    stCoating1 : DUT_PositionState;
    stCoating2 : DUT_PositionState;
END_VAR
VAR_OUTPUT
    {attribute 'pytmc' := '
      pv: GET;
      io: i;
    '}
    enumGet : ENUM_Coating_States;
  END_VAR
VAR
    bCoatingInit : BOOL;
END_VAR

if NOT bCoatingInit THEN
    bCoatingInit := TRUE;

    arrStates[1] := stCoating1;
    arrStates[2] := stCoating2;
END_IF

setState := enumSet;
Exec();
enumGet := getState;
enumSet := setState;

END_FUNCTION_BLOCK

// ---- POUs/Main.TcPOU
PROGRAM Main
VAR
    tpImAPLC : TP := (PT:=T#10S);

    // MR1L3
    // Motors
    {attribute 'TcLinkTo' := '.bLimitForwardEnable:=TIIB[EL7041-1000_M1L3_Yup]^STM Status^Status^Digital input 1;
                              .bLimitBackwardEnable:=TIIB[EL7041-1000_M1L3_Yup]^STM Status^Status^Digital input 2;
                              .nRawEncoderULINT:=TIIB[EL5042_M1L3_Yupdwn]^FB Inputs Channel 1^Position'}
    {attribute 'pytmc' := '
        pv: MR1L3:HOMS:MMS:YUP
    '}
    //PMPS State Stage; bPowerSelf:=False
    M1 : DUT_MotionStage := (sName:='MR1L3-Coatings', fVelocity:=200.0, nEnableMode:=ENUM_StageEnableMode.ALWAYS, bPowerSelf:=FALSE);
    fbMotionStage_m1 : FB_MotionStage;

    {attribute 'TcLinkTo' := '.bLimitForwardEnable:=TIIB[EL7041-1000_M1L3_Ydwn]^STM Status^Status^Digital input 1;
                              .bLimitBackwardEnable:=TIIB[EL7041-1000_M1L3_Ydwn]^STM Status^Status^Digital input 2'}
    {attribute 'pytmc' := '
        pv: MR1L3:HOMS:MMS:YDWN
    '}
    M2 : DUT_MotionStage := (fVelocity:=200.0, nEnableMode:=ENUM_StageEnableMode.ALWAYS, bPowerSelf:=TRUE);
    fbMotionStage_m2 : FB_MotionStage;

    {attribute 'TcLinkTo' := '.bLimitForwardEnable:=TIIB[EL7041-1000_M1L3_Xup]^STM Status^Status^Digital input 1;
                              .bLimitBackwardEnable:=TIIB[EL7041-1000_M1L3_Xup]^STM Status^Status^Digital input 2;
                              .nRawEncoderULINT:=TIIB[EL5042_M1L3_Xupdwn]^FB Inputs Channel 1^Position'}
    {attribute 'pytmc' := '
        pv: MR1L3:HOMS:MMS:XUP
    '}
    M3 : DUT_MotionStage := (fVelocity:=1000.0, nEnableMode:=ENUM_StageEnableMode.ALWAYS, bPowerSelf:=TRUE);
    fbMotionStage_m3 : FB_MotionStage;

    {attribute 'TcLinkTo' := '.bLimitForwardEnable:=TIIB[EL7041-1000_M1L3_Xdwn]^STM Status^Status^Digital input 1;
                              .bLimitBackwardEnable:=TIIB[EL7041-1000_M1L3_Xdwn]^STM Status^Status^Digital input 2'}
    {attribute 'pytmc' := '
        pv: MR1L3:HOMS:MMS:XDWN
    '}
    M4 : DUT_MotionStage := (fVelocity:=1000.0, nEnableMode:=ENUM_StageEnableMode.ALWAYS, bPowerSelf:=TRUE);
    fbMotionStage_m4 : FB_MotionStage;

    {attribute 'TcLinkTo' := '.bLimitForwardEnable:=TIIB[EL7041-1000_M1L3_PitchCoarse]^STM Status^Status^Digital input 1;
                              .bLimitBackwardEnable:=TIIB[EL7041-1000_M1L3_PitchCoarse]^STM Status^Status^Digital input 2;
                              .nRawEncoderULINT:=TIIB[EL5042_M1L3_PitchBender]^FB Inputs Channel 1^Position'}
    {attribute 'pytmc' := '
        pv: MR1L3:HOMS:MMS:PITCH
    '}
    M5 : DUT_MotionStage := (fVelocity:=150.0, nEnableMode:=ENUM_StageEnableMode.ALWAYS, bPowerSelf:=TRUE); // MR1L3 Pitch Stepper
    fbMotionStage_m5 : FB_MotionStage;

    {attribute 'TcLinkTo' := '.bLimitForwardEnable:=TIIB[EL7041-1000_M1L3_Bender]^STM Status^Status^Digital input 1;
                              .bLimitBackwardEnable:=TIIB[EL7041-1000_M1L3_Bender]^STM Status^Status^Digital input 2;
                              .nRawEncoderULINT:=TIIB[EL5042_M1L3_PitchBender]^FB Inputs Channel 2^Position'}
    {attribute 'pytmc' := '
        pv: MR1L3:HOMS:MMS:BENDER
    '}
    M6 : DUT_MotionStage := (fVelocity:=150.0, nEnableMode:=ENUM_StageEnableMode.ALWAYS, bPowerSelf:=TRUE); // MR1L3 Bender
    fbMotionStage_m6 : FB_MotionStage;

    {attribute 'TcLinkTo' := '.fbRunHOMS.bSTOEnable1:=TIIB[EL1004_M1L3_STO]^Channel 1^Input;
                              .fbRunHOMS.bSTOEnable2:=TIIB[EL1004_M1L3_STO]^Channel 2^Input;
                              .fbRunHOMS.stYupEnc.Count:=TIIB[EL5042_M1L3_Yupdwn]^FB Inputs Channel 1^Position;
                              .fbRunHOMS.stYdwnEnc.Count:=TIIB[EL5042_M1L3_Yupdwn]^FB Inputs Channel 2^Position;
                              .fbRunHOMS.stXupEnc.Count:=TIIB[EL5042_M1L3_Xupdwn]^FB Inputs Channel 1^Position;
                              .fbRunHOMS.stXdwnEnc.Count:=TIIB[EL5042_M1L3_Xupdwn]^FB Inputs Channel 2^Position'}
    {attribute 'pytmc' := '
        pv: MR1L3:HOMS
    '}
    MR1L3 : DUT_HOMS;
    {attribute 'pytmc' := '
        pv: MR1L3:HOMS:STATS
    '}
    fbMR1L3GantryStats : FB_HomsStats;

    // Encoder Arrays/RMS Watch:
    {attribute 'pytmc' := '
        pv: MR1L3:HOMS:ENC:Y
    '}
    fbYRMSErrorMR1L3 : FB_RMSWatch;
    fMaxYRMSErrorMR1L3 : LREAL;
    fMinYRMSErrorMR1L3 : LREAL;

    {attribute 'pytmc' := '
        pv: MR1L3:HOMS:ENC:X
    '}
    fbXRMSErrorMR1L3 : FB_RMSWatch;
    fMaxXRMSErrorMR1L3 : LREAL;
    fMinXRMSErrorMR1L3 : LREAL;

    {attribute 'pytmc' := '
        pv: MR1L3:HOMS:ENC:PITCH
    '}
    fbPitchRMSErrorMR1L3 : FB_RMSWatch;
    fMaxPitchRMSErrorMR1L3 : LREAL;
    fMinPitchRMSErrorMR1L3 : LREAL;

    {attribute 'pytmc' := '
        pv: MR1L3:HOMS:ENC:BENDER
    '}
    fbBenderRMSErrorMR1L3 : FB_RMSWatch;
    fMaxBenderRMSErrorMR1L3 : LREAL;
    fMinBenderRMSErrorMR1L3 : LREAL;

    // Pitch Control
    fbMR1L3PitchControl : FB_PitchControl;
    bMR1L3PitchDone : BOOL;
    bMR1L3PitchBusy : BOOL;

    // Bender Control
    fbBenderMR1L3 : FB_Bender;

    // Raw Encoder Counts
    {attribute 'pytmc' := '
        pv: MR1L3:HOMS:ENC:YUP:CNT
        field: EGU cnt
        io: i
    '}
    nEncCntYupMR1L3 : UDINT;
    {attribute 'pytmc' := '
        pv: MR1L3:HOMS:ENC:YDWN:CNT
        field: EGU cnt
        io: i
    '}
    nEncCntYdwnMR1L3 : UDINT;
    {attribute 'pytmc' := '
        pv: MR1L3:HOMS:ENC:XUP:CNT
        field: EGU cnt
        io: i
    '}
    nEncCntXupMR1L3 : UDINT;
    {attribute 'pytmc' := '
        pv: MR1L3:HOMS:ENC:XDWN:CNT
        field: EGU cnt
        io: i
    '}
    nEncCntXdwnMR1L3 : UDINT;
    {attribute 'pytmc' := '
        pv: MR1L3:HOMS:ENC:PITCH:CNT
        field: EGU cnt
        io: i
    '}
    nEncCntPitchMR1L3 : UDINT;

    // Encoder Reference Values
    {attribute 'pytmc' := '
        pv: MR1L3:HOMS:ENC:YUP:REF
        field: EGU cnt
        io: i
    '}
    nEncRefYupMR1L3 : UDINT;
    {attribute 'pytmc' := '
        pv: MR1L3:HOMS:ENC:YDWN:REF
        field: EGU cnt
        io: i
    '}
    nEncRefYdwnMR1L3 : UDINT;
    {attribute 'pytmc' := '
        pv: MR1L3:HOMS:ENC:XUP:REF
        field: EGU cnt
        io: i
    '}
    nEncRefXupMR1L3 : UDINT;
    {attribute 'pytmc' := '
        pv: MR1L3:HOMS:ENC:XDWN:REF
        field: EGU cnt
        io: i
    '}
    nEncRefXdwnMR1L3 : UDINT;
    {attribute 'pytmc' := '
        pv: MR1L3:HOMS:ENC:PITCH:REF
        field: EGU cnt
        io: i
    '}
    nEncRefPitchMR1L3 : UDINT;
    mcReadParameterPitchMR1L3 : MC_ReadParameter;
    fEncRefPitchMR1L3_urad : LREAL; // Current Pitch encoder offset in urad
    // MR1L4
    // Motors
    {attribute 'TcLinkTo' := '.bLimitForwardEnable:=TIIB[EL7041-1000_M1L4_Yup]^STM Status^Status^Digital input 1;
                              .bLimitBackwardEnable:=TIIB[EL7041-1000_M1L4_Yup]^STM Status^Status^Digital input 2;
                              .nRawEncoderULINT:=TIIB[EL5042_M1L4_Yupdwn]^FB Inputs Channel 1^Position'}
    {attribute 'pytmc' := '
        pv: MR1L4:HOMS:MMS:YUP
    '}
    M7 : DUT_MotionStage := (fVelocity:=200.0, nEnableMode:=ENUM_StageEnableMode.ALWAYS, bPowerSelf:=TRUE);
    fbMotionStage_m7 : FB_MotionStage;
    {attribute 'TcLinkTo' := '.bLimitForwardEnable:=TIIB[EL7041-1000_M1L4_Ydwn]^STM Status^Status^Digital input 1;
                              .bLimitBackwardEnable:=TIIB[EL7041-1000_M1L4_Ydwn]^STM Status^Status^Digital input 2'}
    {attribute 'pytmc' := '
        pv: MR1L4:HOMS:MMS:YDWN
    '}
    M8 : DUT_MotionStage := (fVelocity:=200.0, nEnableMode:=ENUM_StageEnableMode.ALWAYS, bPowerSelf:=TRUE);
    fbMotionStage_m8 : FB_MotionStage;
    {attribute 'TcLinkTo' := '.bLimitForwardEnable:=TIIB[EL7041-1000_M1L4_Xup]^STM Status^Status^Digital input 1;
                              .bLimitBackwardEnable:=TIIB[EL7041-1000_M1L4_Xup]^STM Status^Status^Digital input 2;
                              .nRawEncoderULINT:=TIIB[EL5042_M1L4_Xupdwn]^FB Inputs Channel 1^Position'}
    {attribute 'pytmc' := '
        pv: MR1L4:HOMS:MMS:XUP
    '}
    M9 : DUT_MotionStage := (fVelocity:=1000.0, nEnableMode:=ENUM_StageEnableMode.ALWAYS, bPowerSelf:=TRUE);
    fbMotionStage_m9 : FB_MotionStage;
    {attribute 'TcLinkTo' := '.bLimitForwardEnable:=TIIB[EL7041-1000_M1L4_Xdwn]^STM Status^Status^Digital input 1;
                              .bLimitBackwardEnable:=TIIB[EL7041-1000_M1L4_Xdwn]^STM Status^Status^Digital input 2'}
    {attribute 'pytmc' := '
        pv: MR1L4:HOMS:MMS:XDWN
    '}
    M10 : DUT_MotionStage := (fVelocity:=1000.0, nEnableMode:=ENUM_StageEnableMode.ALWAYS, bPowerSelf:=TRUE);
    fbMotionStage_m10 : FB_MotionStage;
    {attribute 'TcLinkTo' := '.bLimitForwardEnable:=TIIB[EL7041-1000_M1L4_PitchCoarse]^STM Status^Status^Digital input 1;
                              .bLimitBackwardEnable:=TIIB[EL7041-1000_M1L4_PitchCoarse]^STM Status^Status^Digital input 2;
                              .nRawEncoderULINT:=TIIB[EL5042_M1L4_PitchBender]^FB Inputs Channel 1^Position'}
    {attribute 'pytmc' := '
        pv: MR1L4:HOMS:MMS:PITCH
    '}
    M11 : DUT_MotionStage := (fVelocity:=150.0, nEnableMode:=ENUM_StageEnableMode.ALWAYS, bPowerSelf:=TRUE); // MR1L4 Pitch Stepper
    fbMotionStage_m11 : FB_MotionStage;
    {attribute 'TcLinkTo' := '.bLimitForwardEnable:=TIIB[EL7041-1000_M1L4_Bender]^STM Status^Status^Digital input 1;
                              .bLimitBackwardEnable:=TIIB[EL7041-1000_M1L4_Bender]^STM Status^Status^Digital input 2;
                              .nRawEncoderULINT:=TIIB[EL5042_M1L4_PitchBender]^FB Inputs Channel 2^Position'}
    {attribute 'pytmc' := '
        pv: MR1L4:HOMS:MMS:BENDER
    '}
    M12 : DUT_MotionStage := (fVelocity:=150.0, nEnableMode:=ENUM_StageEnableMode.ALWAYS, bPowerSelf:=TRUE); // MR1L4 Bender
    fbMotionStage_m12 : FB_MotionStage;
    {attribute 'TcLinkTo' := '.fbRunHOMS.bSTOEnable1:=TIIB[EL1004_M1L4_STO]^Channel 1^Input;
                              .fbRunHOMS.bSTOEnable2:=TIIB[EL1004_M1L4_STO]^Channel 2^Input;
                              .fbRunHOMS.stYupEnc.Count:=TIIB[EL5042_M1L4_Yupdwn]^FB Inputs Channel 1^Position;
                              .fbRunHOMS.stYdwnEnc.Count:=TIIB[EL5042_M1L4_Yupdwn]^FB Inputs Channel 2^Position;
                              .fbRunHOMS.stXupEnc.Count:=TIIB[EL5042_M1L4_Xupdwn]^FB Inputs Channel 1^Position;
                              .fbRunHOMS.stXdwnEnc.Count:=TIIB[EL5042_M1L4_Xupdwn]^FB Inputs Channel 2^Position'}
    {attribute 'pytmc' := '
        pv: MR1L4:HOMS
    '}
    MR1L4 : DUT_HOMS;
    {attribute 'pytmc' := '
        pv: MR1L4:HOMS:STATS
    '}
    fbMR1L4GantryStats : FB_HomsStats;
    // Encoder Arrays/RMS Watch:
    {attribute 'pytmc' := '
        pv: MR1L4:HOMS:ENC:Y
    '}
    fbYRMSErrorMR1L4 : FB_RMSWatch;
    fMaxYRMSErrorMR1L4 : LREAL;
    fMinYRMSErrorMR1L4 : LREAL;

    {attribute 'pytmc' := '
        pv: MR1L4:HOMS:ENC:X
    '}
    fbXRMSErrorMR1L4 : FB_RMSWatch;
    fMaxXRMSErrorMR1L4 : LREAL;
    fMinXRMSErrorMR1L4 : LREAL;

    {attribute 'pytmc' := '
        pv: MR1L4:HOMS:ENC:PITCH
    '}
    fbPitchRMSErrorMR1L4 : FB_RMSWatch;
    fMaxPitchRMSErrorMR1L4 : LREAL;
    fMinPitchRMSErrorMR1L4 : LREAL;

    {attribute 'pytmc' := '
        pv: MR1L4:HOMS:ENC:BENDER
    '}
    fbBenderRMSErrorMR1L4 : FB_RMSWatch;
    fMaxBenderRMSErrorMR1L4 : LREAL;
    fMinBenderRMSErrorMR1L4 : LREAL;

    // Pitch Control
    fbMR1L4PitchControl : FB_PitchControl;
    bMR1L4PitchDone : BOOL;
    bMR1L4PitchBusy : BOOL;

    // Bender Control
    fbBenderMR1L4 : FB_Bender;

    // Raw Encoder Counts
    {attribute 'pytmc' := '
        pv: MR1L4:HOMS:ENC:YUP:CNT
        field: EGU cnt
        io: i
    '}
    nEncCntYupMR1L4 : UDINT;
    {attribute 'pytmc' := '
        pv: MR1L4:HOMS:ENC:YDWN:CNT
        field: EGU cnt
        io: i
    '}
    nEncCntYdwnMR1L4 : UDINT;
    {attribute 'pytmc' := '
        pv: MR1L4:HOMS:ENC:XUP:CNT
        field: EGU cnt
        io: i
    '}
    nEncCntXupMR1L4 : UDINT;
    {attribute 'pytmc' := '
        pv: MR1L4:HOMS:ENC:XDWN:CNT
        field: EGU cnt
        io: i
    '}
    nEncCntXdwnMR1L4 : UDINT;
    {attribute 'pytmc' := '
        pv: MR1L4:HOMS:ENC:PITCH:CNT
        field: EGU cnt
        io: i
    '}
    nEncCntPitchMR1L4 : UDINT;

    // Encoder Reference Values
    {attribute 'pytmc' := '
        pv: MR1L4:HOMS:ENC:YUP:REF
        field: EGU cnt
        io: i
    '}
    nEncRefYupMR1L4 : UDINT;
    {attribute 'pytmc' := '
        pv: MR1L4:HOMS:ENC:YDWN:REF
        field: EGU cnt
        io: i
    '}
    nEncRefYdwnMR1L4 : UDINT;
    {attribute 'pytmc' := '
        pv: MR1L4:HOMS:ENC:XUP:REF
        field: EGU cnt
        io: i
    '}
    nEncRefXupMR1L4 : UDINT;
    {attribute 'pytmc' := '
        pv: MR1L4:HOMS:ENC:XDWN:REF
        field: EGU cnt
        io: i
    '}
    nEncRefXdwnMR1L4 : UDINT;
    {attribute 'pytmc' := '
        pv: MR1L4:HOMS:ENC:PITCH:REF
        field: EGU cnt
        io: i
    '}
    nEncRefPitchMR1L4 : UDINT;
    mcReadParameterPitchMR1L4 : MC_ReadParameter;
    fEncRefPitchMR1L4_urad : LREAL; // Current Pitch encoder offset in urad

// MR2L3 BECKHOFF
// Motors
    {attribute 'TcLinkTo' := '.bLimitForwardEnable:=TIIB[EL7041-1000_M2L3_Yup]^STM Status^Status^Digital input 1;
                              .bLimitBackwardEnable:=TIIB[EL7041-1000_M2L3_Yup]^STM Status^Status^Digital input 2';
                              .nRawEncoderULINT:=TIIB[EL5042_M2L3_Yupdwn]^FB Inputs Channel 1^Position'}
    {attribute 'pytmc' := '
        pv: MR2L3:HOMS:MMS:YUP
    '}
    M13 : DUT_MotionStage := (fVelocity:=200.0, nEnableMode:=ENUM_StageEnableMode.ALWAYS, bPowerSelf:=TRUE); // MR2L3 Yup
    fbMotionStage_m13 : FB_MotionStage;


    {attribute 'TcLinkTo' := '.bLimitForwardEnable:=TIIB[EL7041-1000_M2L3_Ydwn]^STM Status^Status^Digital input 1;
                              .bLimitBackwardEnable:=TIIB[EL7041-1000_M2L3_Ydwn]^STM Status^Status^Digital input 2'}
    {attribute 'pytmc' := '
        pv: MR2L3:HOMS:MMS:YDWN
    '}
    M14 : DUT_MotionStage := (fVelocity:=200.0, nEnableMode:=ENUM_StageEnableMode.ALWAYS, bPowerSelf:=TRUE); // MR2L3 Ydwn
    fbMotionStage_m14 : FB_MotionStage;

    {attribute 'TcLinkTo' := '.bLimitForwardEnable:=TIIB[EL7041-1000_M2L3_Xup]^STM Status^Status^Digital input 1;
                              .bLimitBackwardEnable:=TIIB[EL7041-1000_M2L3_Xup]^STM Status^Status^Digital input 2;
                              .nRawEncoderULINT:=TIIB[EL5042_M2L3_Xupdwn]^FB Inputs Channel 1^Position'}
    {attribute 'pytmc' := '
        pv: MR2L3:HOMS:MMS:XUP
    '}
    M15 : DUT_MotionStage := (fVelocity:=1000.0, nEnableMode:=ENUM_StageEnableMode.ALWAYS, bPowerSelf:=TRUE); // MR2L3 Xup
    fbMotionStage_m15 : FB_MotionStage;

    {attribute 'TcLinkTo' := '.bLimitForwardEnable:=TIIB[EL7041-1000_M2L3_Xdwn]^STM Status^Status^Digital input 1;
                              .bLimitBackwardEnable:=TIIB[EL7041-1000_M2L3_Xdwn]^STM Status^Status^Digital input 2'}
    {attribute 'pytmc' := '
        pv: MR2L3:HOMS:MMS:XDWN
    '}
    M16 : DUT_MotionStage := (fVelocity:=1000.0, nEnableMode:=ENUM_StageEnableMode.ALWAYS, bPowerSelf:=TRUE); // MR2L3 Xdwn
    fbMotionStage_m16 : FB_MotionStage;

    {attribute 'TcLinkTo' := '.bLimitForwardEnable:=TIIB[EL7041-1000_M2L3_PitchCoarse]^STM Status^Status^Digital input 1;
                              .bLimitBackwardEnable:=TIIB[EL7041-1000_M2L3_PitchCoarse]^STM Status^Status^Digital input 2;
                              .nRawEncoderULINT:=TIIB[EL5042_M2L3_PitchBender]^FB Inputs Channel 1^Position'}
    {attribute 'pytmc' := '
        pv: MR2L3:HOMS:MMS:PITCH
    '}
    M17 : DUT_MotionStage := (fVelocity:=150.0, nEnableMode:=ENUM_StageEnableMode.ALWAYS, bPowerSelf:=TRUE); // MR2L3 Pitch Stepper
    fbMotionStage_m17 : FB_MotionStage;
    {attribute 'TcLinkTo' := '.bLimitForwardEnable:=TIIB[EL7041-1000_M2L3_Bender]^STM Status^Status^Digital input 1;
                              .bLimitBackwardEnable:=TIIB[EL7041-1000_M2L3_Bender]^STM Status^Status^Digital input 2;
                              .nRawEncoderULINT:=TIIB[EL5042_M2L3_PitchBender]^FB Inputs Channel 2^Position'}
    {attribute 'pytmc' := '
        pv: MR2L3:HOMS:MMS:BENDER
    '}
    M18 : DUT_MotionStage := (fVelocity:=150.0, nEnableMode:=ENUM_StageEnableMode.ALWAYS, bPowerSelf:=TRUE); // MR2L3 Bender
    fbMotionStage_m18 : FB_MotionStage;

    {attribute 'TcLinkTo' := '.fbRunHOMS.bSTOEnable1:=TIIB[EL1004_M2L3_STO]^Channel 1^Input;
                              .fbRunHOMS.bSTOEnable2:=TIIB[EL1004_M2L3_STO]^Channel 2^Input;
                              .fbRunHOMS.stYupEnc.Count:=TIIB[EL5042_M2L3_Yupdwn]^FB Inputs Channel 1^Position;
                              .fbRunHOMS.stYdwnEnc.Count:=TIIB[EL5042_M2L3_Yupdwn]^FB Inputs Channel 2^Position;
                              .fbRunHOMS.stXupEnc.Count:=TIIB[EL5042_M2L3_Xupdwn]^FB Inputs Channel 1^Position;
                              .fbRunHOMS.stXdwnEnc.Count:=TIIB[EL5042_M2L3_Xupdwn]^FB Inputs Channel 2^Position'}
    {attribute 'pytmc' := '
        pv: MR2L3:HOMS
    '}
    MR2L3 : DUT_HOMS;
    {attribute 'pytmc' := '
        pv: MR2L3:HOMS:STATS
    '}
    fbMR2L3GantryStats : FB_HomsStats;

    // Encoder Arrays/RMS Watch:
    {attribute 'pytmc' := '
        pv: MR2L3:HOMS:ENC:Y
    '}
    fbYRMSErrorMR2L3 : FB_RMSWatch;
    fMaxYRMSErrorMR2L3 : LREAL;
    fMinYRMSErrorMR2L3 : LREAL;

    {attribute 'pytmc' := '
        pv: MR2L3:HOMS:ENC:X
    '}
    fbXRMSErrorMR2L3 : FB_RMSWatch;
    fMaxXRMSErrorMR2L3 : LREAL;
    fMinXRMSErrorMR2L3 : LREAL;

    {attribute 'pytmc' := '
        pv: MR2L3:HOMS:ENC:PITCH
    '}
    fbPitchRMSErrorMR2L3 : FB_RMSWatch;
    fMaxPitchRMSErrorMR2L3 : LREAL;
    fMinPitchRMSErrorMR2L3 : LREAL;

    {attribute 'pytmc' := '
        pv: MR2L3:HOMS:ENC:BENDER
    '}
    fbBenderRMSErrorMR2L3 : FB_RMSWatch;
    fMaxBenderRMSErrorMR2L3 : LREAL;
    fMinBenderRMSErrorMR2L3 : LREAL;

    // Pitch Control
    fbMR2L3PitchControl : FB_PitchControl;
    bMR2L3PitchDone : BOOL;
    bMR2L3PitchBusy : BOOL;

    // Bender Control
    fbBenderMR2L3 : FB_Bender;

    // Raw Encoder Counts
    {attribute 'pytmc' := '
        pv: MR2L3:HOMS:ENC:YUP:CNT
        field: EGU cnt
        io: i
    '}
    nEncCntYupMR2L3 : UDINT;
    {attribute 'pytmc' := '
        pv: MR2L3:HOMS:ENC:YDWN:CNT
        field: EGU cnt
        io: i
    '}
    nEncCntYdwnMR2L3 : UDINT;
    {attribute 'pytmc' := '
        pv: MR2L3:HOMS:ENC:XUP:CNT
        field: EGU cnt
        io: i
    '}
    nEncCntXupMR2L3 : UDINT;
    {attribute 'pytmc' := '
        pv: MR2L3:HOMS:ENC:XDWN:CNT
        field: EGU cnt
        io: i
    '}
    nEncCntXdwnMR2L3 : UDINT;
    {attribute 'pytmc' := '
        pv: MR2L3:HOMS:ENC:PITCH:CNT
        field: EGU cnt
        io: i
    '}
    nEncCntPitchMR2L3 : UDINT;

    // Encoder Reference Values
    {attribute 'pytmc' := '
        pv: MR2L3:HOMS:ENC:YUP:REF
        field: EGU cnt
        io: i
    '}
    nEncRefYupMR2L3 : UDINT;
    {attribute 'pytmc' := '
        pv: MR2L3:HOMS:ENC:YDWN:REF
        field: EGU cnt
        io: i
    '}
    nEncRefYdwnMR2L3 : UDINT;
    {attribute 'pytmc' := '
        pv: MR2L3:HOMS:ENC:XUP:REF
        field: EGU cnt
        io: i
    '}
    nEncRefXupMR2L3 : UDINT;
    {attribute 'pytmc' := '
        pv: MR2L3:HOMS:ENC:XDWN:REF
        field: EGU cnt
        io: i
    '}
    nEncRefXdwnMR2L3 : UDINT;
    {attribute 'pytmc' := '
        pv: MR2L3:HOMS:ENC:PITCH:REF
        field: EGU cnt
        io: i
    '}
    nEncRefPitchMR2L3 : UDINT;
    mcReadParameterPitchMR2L3 : MC_ReadParameter;
    fEncRefPitchMR2L3_urad : LREAL; // Current Pitch encoder offset in urad


    // Common
    fEncLeverArm_mm : LREAL := 513.0;

    // Logging
    fbLogHandler : FB_LogHandler;
END_VAR

// MR1L3 BECKHOFF
MR1L3.fbRunHOMS(stYup:=M1,
               stYdwn:=M2,
               stXup:=M3,
               stXdwn:=M4,
               stPitch:=M5,
               nYupEncRef:=GVL_MR1L3_Constants.nYUP_ENC_REF,
               nYdwnEncRef:=GVL_MR1L3_Constants.nYDWN_ENC_REF,
               nXupEncRef:=GVL_MR1L3_Constants.nXUP_ENC_REF,
               nXdwnEncRef:=GVL_MR1L3_Constants.nXDWN_ENC_REF,
               bExecuteCoupleY:=MR1L3.bExecuteCoupleY,
               bExecuteCoupleX:=MR1L3.bExecuteCoupleX,
               bExecuteDecoupleY:=MR1L3.bExecuteDecoupleY,
               bExecuteDecoupleX:=MR1L3.bExecuteDecoupleX,
               bGantryAlreadyCoupledY=>MR1L3.bGantryAlreadyCoupledY,
               bGantryAlreadyCoupledX=>MR1L3.bGantryAlreadyCoupledX,
               nCurrGantryY=>MR1L3.nCurrGantryY,
               nCurrGantryX=>MR1L3.nCurrGantryX);
fbBenderMR1L3(stBender:=M6,
             bSTOEnable1:=MR1L3.fbRunHOMS.bSTOEnable1,
             bSTOEnable2:=MR1L3.fbRunHOMS.bSTOEnable2);
// No slave motion through Epics
M2.bExecute := FALSE; // MR1L3-Ydwn
M4.bExecute := FALSE; // MR1L3-Xdwn

// Convert nCurrGantry to um (smaller number) to read out in epics
MR1L3.fCurrGantryY_um := LINT_TO_REAL(MR1L3.nCurrGantryY) / 1000.0;
MR1L3.fCurrGantryX_um := LINT_TO_REAL(MR1L3.nCurrGantryX) / 1000.0;

// FB_MotionStage's for non-piezo axes
fbMotionStage_m1(stMotionStage:=M1);
fbMotionStage_m2(stMotionStage:=M2);
fbMotionStage_m3(stMotionStage:=M3);
fbMotionStage_m4(stMotionStage:=M4);
fbMotionStage_m5(stMotionStage:=M5);
fbMotionStage_m6(stMotionStage:=M6);

// Calculate Gantry Stats
fbMR1L3GantryStats(homs:=MR1L3, fbUpStreamY:=M1, fbUpStreamX:=M3);
fbMR1L4GantryStats(homs:=MR1L4, fbUpStreamY:=M7, fbUpStreamX:=M9);
fbMR2L3GantryStats(homs:=MR2L3, fbUpStreamY:=M13, fbUpStreamX:=M15);

// Calculate Pitch RMS Error:
fbYRMSErrorMR1L3(stMotionStage:=M1,
                fMaxRMSError=>fMaxYRMSErrorMR1L3,
                fMinRMSError=>fMinYRMSErrorMR1L3);

fbXRMSErrorMR1L3(stMotionStage:=M3,
                fMaxRMSError=>fMaxXRMSErrorMR1L3,
                fMinRMSError=>fMinXRMSErrorMR1L3);

fbPitchRMSErrorMR1L3(stMotionStage:=M5,
                    fMaxRMSError=>fMaxPitchRMSErrorMR1L3,
                    fMinRMSError=>fMinPitchRMSErrorMR1L3);

fbBenderRMSErrorMR1L3(stMotionStage:=M6,
                     fMaxRMSError=>fMaxBenderRMSErrorMR1L3,
                     fMinRMSError=>fMinBenderRMSErrorMR1L3);
// Pitch Control
//fbMR1L3PitchControl(Pitch:=GVL_M1.MR1L3_Pitch,
                   //Stepper:=M5,
                   //lrCurrentSetpoint:=M5.fPosition,
                   //q_bDone=>bMR1L3PitchDone,
                   //q_bBusy=>bMR1L3PitchBusy);
// When STO hit, need to reset SP
//IF NOT M5.bHardwareEnable THEN
    //M5.fPosition := M5.stAxisStatus.fActPosition;
//END_IF

// Raw Encoder Counts For Epics
nEncCntYupMR1L3 := ULINT_TO_UDINT(MR1L3.fbRunHOMS.stYupEnc.Count);
nEncCntYdwnMR1L3 := ULINT_TO_UDINT(MR1L3.fbRunHOMS.stYdwnEnc.Count);
nEncCntXupMR1L3 := ULINT_TO_UDINT(MR1L3.fbRunHOMS.stXupEnc.Count);
nEncCntXdwnMR1L3 := ULINT_TO_UDINT(MR1L3.fbRunHOMS.stXdwnEnc.Count);
nEncCntPitchMR1L3 := LINT_TO_UDINT(GVL_MR1L3.MR1L3_Pitch.diEncCnt);

// Encoder Reference Values For Epics
nEncRefYupMR1L3 := ULINT_TO_UDINT(GVL_MR1L3_Constants.nYUP_ENC_REF);
nEncRefYdwnMR1L3 := ULINT_TO_UDINT(GVL_MR1L3_Constants.nYDWN_ENC_REF);
nEncRefXupMR1L3 := ULINT_TO_UDINT(GVL_MR1L3_Constants.nXUP_ENC_REF);
nEncRefXdwnMR1L3 := ULINT_TO_UDINT(GVL_MR1L3_Constants.nXDWN_ENC_REF);
mcReadParameterPitchMR1L3(Axis:=M5.Axis,
                         Enable:=TRUE,
                         ParameterNumber:=MC_AxisParameter.AxisEncoderOffset,
                         ReadMode:=READMODE_CYCLIC,
                         Value=>fEncRefPitchMR1L3_urad);

nEncRefPitchMR1L3 := LREAL_TO_UDINT(ABS(fEncRefPitchMR1L3_urad) * fEncLeverArm_mm);

//Beckhoff MR1L4
MR1L4.fbRunHOMS(stYup:=M7,
               stYdwn:=M8,
               stXup:=M9,
               stXdwn:=M10,
               stPitch:=M11,
               nYupEncRef:=GVL_MR1L4_Constants.nYUP_ENC_REF,
               nYdwnEncRef:=GVL_MR1L4_Constants.nYDWN_ENC_REF,
               nXupEncRef:=GVL_MR1L4_Constants.nXUP_ENC_REF,
               nXdwnEncRef:=GVL_MR1L4_Constants.nXDWN_ENC_REF,
               bExecuteCoupleY:=MR1L4.bExecuteCoupleY,
               bExecuteCoupleX:=MR1L4.bExecuteCoupleX,
               bExecuteDecoupleY:=MR1L4.bExecuteDecoupleY,
               bExecuteDecoupleX:=MR1L4.bExecuteDecoupleX,
               bGantryAlreadyCoupledY=>MR1L4.bGantryAlreadyCoupledY,
               bGantryAlreadyCoupledX=>MR1L4.bGantryAlreadyCoupledX,
               nCurrGantryY=>MR1L4.nCurrGantryY,
               nCurrGantryX=>MR1L4.nCurrGantryX);
fbBenderMR1L4(stBender:=M12,
             bSTOEnable1:=MR1L4.fbRunHOMS.bSTOEnable1,
             bSTOEnable2:=MR1L4.fbRunHOMS.bSTOEnable2);
// No slave motion through Epics
M8.bExecute := FALSE; // MR1L3-Ydwn
M10.bExecute := FALSE; // MR1L3-Xdwn

// Convert nCurrGantry to um (smaller number) to read out in epics
MR1L4.fCurrGantryY_um := LINT_TO_REAL(MR1L4.nCurrGantryY) / 1000.0;
MR1L4.fCurrGantryX_um := LINT_TO_REAL(MR1L4.nCurrGantryX) / 1000.0;

// FB_MotionStage's for non-piezo axes
fbMotionStage_m7(stMotionStage:=M7);
fbMotionStage_m8(stMotionStage:=M8);
fbMotionStage_m9(stMotionStage:=M9);
fbMotionStage_m10(stMotionStage:=M10);
fbMotionStage_m11(stMotionStage:=M11);
fbMotionStage_m12(stMotionStage:=M12);

// Calculate Pitch RMS Error:
fbYRMSErrorMR1L4(stMotionStage:=M7,
                fMaxRMSError=>fMaxYRMSErrorMR1L4,
                fMinRMSError=>fMinYRMSErrorMR1L4);

fbXRMSErrorMR1L4(stMotionStage:=M9,
                fMaxRMSError=>fMaxXRMSErrorMR1L4,
                fMinRMSError=>fMinXRMSErrorMR1L4);

fbPitchRMSErrorMR1L4(stMotionStage:=M11,
                    fMaxRMSError=>fMaxPitchRMSErrorMR1L4,
                    fMinRMSError=>fMinPitchRMSErrorMR1L4);

fbBenderRMSErrorMR1L4(stMotionStage:=M12,
                     fMaxRMSError=>fMaxBenderRMSErrorMR1L4,
                     fMinRMSError=>fMinBenderRMSErrorMR1L4);
// Pitch Control
//fbMR1L4PitchControl(Pitch:=GVL_M1L4.MR1L4_Pitch,
                   //Stepper:=M11,
                   //lrCurrentSetpoint:=M11.fPosition,
                   //q_bDone=>bMR1L4PitchDone,
                   //q_bBusy=>bMR1L4PitchBusy);
// When STO hit, need to reset SP
//IF NOT M11.bHardwareEnable THEN
    //M11.fPosition := M11.stAxisStatus.fActPosition;
//END_IF

// Raw Encoder Counts For Epics
nEncCntYupMR1L4 := ULINT_TO_UDINT(MR1L4.fbRunHOMS.stYupEnc.Count);
nEncCntYdwnMR1L4 := ULINT_TO_UDINT(MR1L4.fbRunHOMS.stYdwnEnc.Count);
nEncCntXupMR1L4 := ULINT_TO_UDINT(MR1L4.fbRunHOMS.stXupEnc.Count);
nEncCntXdwnMR1L4 := ULINT_TO_UDINT(MR1L4.fbRunHOMS.stXdwnEnc.Count);
nEncCntPitchMR1L4 := LINT_TO_UDINT(GVL_MR1L4.MR1L4_Pitch.diEncCnt);

// Encoder Reference Values For Epics
nEncRefYupMR1L4 := ULINT_TO_UDINT(GVL_MR1L4_Constants.nYUP_ENC_REF);
nEncRefYdwnMR1L4 := ULINT_TO_UDINT(GVL_MR1L4_Constants.nYDWN_ENC_REF);
nEncRefXupMR1L4 := ULINT_TO_UDINT(GVL_MR1L4_Constants.nXUP_ENC_REF);
nEncRefXdwnMR1L4 := ULINT_TO_UDINT(GVL_MR1L4_Constants.nXDWN_ENC_REF);

mcReadParameterPitchMR1L4(Axis:=M11.Axis,
                         Enable:=TRUE,
                         ParameterNumber:=MC_AxisParameter.AxisEncoderOffset,
                         ReadMode:=READMODE_CYCLIC,
                         Value=>fEncRefPitchMR1L4_urad);

nEncRefPitchMR1L4 := LREAL_TO_UDINT(ABS(fEncRefPitchMR1L4_urad) * fEncLeverArm_mm);

//Beckhoff MR2L3
// MR2L3
MR2L3.fbRunHOMS(stYup:=M13,
               stYdwn:=M14,
               stXup:=M15,
               stXdwn:=M16,
               stPitch:=M17,
               nYupEncRef:=GVL_MR2L3_Constants.nYUP_ENC_REF,
               nYdwnEncRef:=GVL_MR2L3_Constants.nYDWN_ENC_REF,
               nXupEncRef:=GVL_MR2L3_Constants.nXUP_ENC_REF,
               nXdwnEncRef:=GVL_MR2L3_Constants.nXDWN_ENC_REF,
               bExecuteCoupleY:=MR2L3.bExecuteCoupleY,
               bExecuteCoupleX:=MR2L3.bExecuteCoupleX,
               bExecuteDecoupleY:=MR2L3.bExecuteDecoupleY,
               bExecuteDecoupleX:=MR2L3.bExecuteDecoupleX,
               bGantryAlreadyCoupledY=>MR2L3.bGantryAlreadyCoupledY,
               bGantryAlreadyCoupledX=>MR2L3.bGantryAlreadyCoupledX,
               nCurrGantryY=>MR2L3.nCurrGantryY,
               nCurrGantryX=>MR2L3.nCurrGantryX);
fbBenderMR2L3(stBender:=M18,
             bSTOEnable1:=MR2L3.fbRunHOMS.bSTOEnable1,
             bSTOEnable2:=MR2L3.fbRunHOMS.bSTOEnable2);
// No slave motion through Epics
M14.bExecute := FALSE; // MR2L3-Ydwn
M16.bExecute := FALSE; // MR2L3-Xdwn

// Convert nCurrGantry to um (smaller number) to read out in epics
MR2L3.fCurrGantryY_um := LINT_TO_REAL(MR2L3.nCurrGantryY) / 1000;
MR2L3.fCurrGantryX_um := LINT_TO_REAL(MR2L3.nCurrGantryX) / 1000;

// FB_MotionStage's for non-piezo axes
fbMotionStage_m13(stMotionStage:=M13);
fbMotionStage_m14(stMotionStage:=M14);
fbMotionStage_m15(stMotionStage:=M15);
fbMotionStage_m16(stMotionStage:=M16);
fbMotionStage_m17(stMotionStage:=M17);
fbMotionStage_m18(stMotionStage:=M18);

// Calculate RMS Error:
fbYRMSErrorMR2L3(stMotionStage:=M13,
                fMaxRMSError=>fMaxYRMSErrorMR2L3,
                fMinRMSError=>fMinYRMSErrorMR2L3);

fbXRMSErrorMR2L3(stMotionStage:=M15,
                fMaxRMSError=>fMaxXRMSErrorMR2L3,
                fMinRMSError=>fMinXRMSErrorMR2L3);

fbPitchRMSErrorMR2L3(stMotionStage:=M17,
                    fMaxRMSError=>fMaxPitchRMSErrorMR2L3,
                    fMinRMSError=>fMinPitchRMSErrorMR2L3);

fbBenderRMSErrorMR2L3(stMotionStage:=M18,
                     fMaxRMSError=>fMaxBenderRMSErrorMR2L3,
                     fMinRMSError=>fMinBenderRMSErrorMR2L3);

// Pitch Control
//fbMR2L3PitchControl(Pitch:=GVL_MR2L3.MR2L3_Pitch,
                   //Stepper:=M17,
                   //lrCurrentSetpoint:=M17.fPosition,
                   //q_bDone=>bMR2L3PitchDone,
                   //q_bBusy=>bMR2L3PitchBusy);
// When STO hit, need to reset SP
//IF NOT M17.bHardwareEnable THEN
    //M17.fPosition := M17.stAxisStatus.fActPosition;
//END_IF

// Raw Encoder Counts For Epics
nEncCntYupMR2L3 := ULINT_TO_UDINT(MR2L3.fbRunHOMS.stYupEnc.Count);
nEncCntYdwnMR2L3 := ULINT_TO_UDINT(MR2L3.fbRunHOMS.stYdwnEnc.Count);
nEncCntXupMR2L3 := ULINT_TO_UDINT(MR2L3.fbRunHOMS.stXupEnc.Count);
nEncCntXdwnMR2L3 := ULINT_TO_UDINT(MR2L3.fbRunHOMS.stXdwnEnc.Count);
nEncCntPitchMR2L3 := LINT_TO_UDINT(GVL_MR2L3.MR2L3_Pitch.diEncCnt);

// Encoder Reference Values For Epics
nEncRefYupMR2L3 := ULINT_TO_UDINT(GVL_MR2L3_Constants.nYUP_ENC_REF);
nEncRefYdwnMR2L3 := ULINT_TO_UDINT(GVL_MR2L3_Constants.nYDWN_ENC_REF);
nEncRefXupMR2L3 := ULINT_TO_UDINT(GVL_MR2L3_Constants.nXUP_ENC_REF);
nEncRefXdwnMR2L3 := ULINT_TO_UDINT(GVL_MR2L3_Constants.nXDWN_ENC_REF);
mcReadParameterPitchMR2L3(Axis:=M17.Axis,
                         Enable:=TRUE,
                         ParameterNumber:=MC_AxisParameter.AxisEncoderOffset,
                         ReadMode:=READMODE_CYCLIC,
                         Value=>fEncRefPitchMR2L3_urad);

nEncRefPitchMR2L3 := LREAL_TO_UDINT(ABS(fEncRefPitchMR2L3_urad) * fEncLeverArm_mm);

bXRT_M2_IN  := Main.MR1L4.fbRunHOMS.stXupEnc.Count < 25490840;
bXRT_M2_OUT := not bXRT_M2_IN;
//States
PRG_States();
//PMPS
PRG_CoatingProtection();
PRG_PMPS();

// Logging
fbLogHandler();

GVL_RTDS.fbMR1L3_Env_RTD_1(fResolution:=0.01);
GVL_RTDS.fbMR1L3_Env_RTD_2(fResolution:=0.01);
GVL_RTDS.fbMR1L3_Env_RTD_3(fResolution:=0.01);

GVL_RTDS.fbMR2L3_Env_RTD_1(fResolution:=0.01);
GVL_RTDS.fbMR2L3_Env_RTD_2(fResolution:=0.01);
GVL_RTDS.fbMR2L3_Env_RTD_3(fResolution:=0.01);

GVL_RTDS.fbMR1L4_Env_RTD_1(fResolution:=0.01);
GVL_RTDS.fbMR1L4_Env_RTD_2(fResolution:=0.01);
GVL_RTDS.fbMR1L4_Env_RTD_3(fResolution:=0.01);

END_PROGRAM

// ---- POUs/PRG_States.TcPOU
PROGRAM PRG_States
VAR
    //MR1L3 Coating States
     {attribute 'pytmc' := '
        pv: MR1L3:HOMS:COATING:STATE;
        io: io;
     '}
    fbMR1L3_Coating_States: FB_Coating_States;

    MR1L3_SiC : DUT_PositionState := (
        bUseRawCounts := TRUE,
        bMoveOk := TRUE,
        bValid := TRUE,
        sName := 'SiC',
        nEncoderCount := 8611100,
        fDelta := 1000,
        fVelocity := 150,
        stBeamParams := PMPS_GVL.cstFullBeam,
        nRequestAssertionID := 16#FA72);

    MR1L3_W : DUT_PositionState := (
        bUseRawCounts := TRUE,
        bMoveOk := TRUE,
        bValid := TRUE,
        sName := 'W',
        nEncoderCount := 18611220,
        fDelta := 1000,
        fVelocity := 150,
        stBeamParams := PMPS_GVL.cstFullBeam,
        nRequestAssertionID := 16#FA73);

//MR1L3 In Out States
    {attribute 'pytmc' := '
        pv: MR1L3:HOMS:MMS:XUP:STATE;
    '}
    fbMR1L3_InOut_States : FB_PositionStateInOut;

    MR1L3_In : DUT_PositionState := (
        bUseRawCounts := TRUE,
        bMoveOk := TRUE,
        bValid := TRUE,
        sName := 'IN',
        nEncoderCount := 25210740,
        fDelta := 1000,
        fVelocity := 150);

    MR1L3_Out : DUT_PositionState := (
        bUseRawCounts := TRUE,
        bMoveOk := TRUE,
        bValid := TRUE,
        sName := 'OUT',
        nEncoderCount := 19210590,
        fDelta := 1000,
        fVelocity := 150);

//MR2L3 Coating States
    {attribute 'pytmc' := '
        pv: MR2L3:HOMS:COATING:STATE;
        io: io;
    '}
    fbMR2L3_Coating_States: FB_Coating_States_noPMPS;

    MR2L3_SiC : DUT_PositionState := (
        bUseRawCounts := TRUE,
        bMoveOk := TRUE,
        bValid := TRUE,
        sName := 'SiC',
        nEncoderCount := 9278970,
        fDelta := 1000,
        fVelocity := 150);

    MR2L3_W : DUT_PositionState := (
        bUseRawCounts := TRUE,
        bMoveOk := TRUE,
        bValid := TRUE,
        sName := 'W',
        nEncoderCount := 19279260,
        fDelta := 1000,
        fVelocity := 150);

//MR1L4 Coating States
    {attribute 'pytmc' := '
        pv: MR1L4:HOMS:COATING:STATE;
        io: io;
    '}
    fbMR1L4_Coating_States: FB_Coating_States_noPMPS;

    MR1L4_SiC : DUT_PositionState := (
        bUseRawCounts := TRUE,
        bMoveOk := TRUE,
        bValid := TRUE,
        sName := 'SiC',
        nEncoderCount := 8495750,
        fDelta := 1000,
        fVelocity := 150);

    MR1L4_W : DUT_PositionState := (
        bUseRawCounts := TRUE,
        bMoveOk := TRUE,
        bValid := TRUE,
        sName := 'W',
        nEncoderCount := 18496280,
        fDelta := 1000,
        fVelocity := 150);

//MR1L4 In Out States
    {attribute 'pytmc' := '
        pv: MR1L4:HOMS:MMS:XUP:STATE;
    '}
    fbMR1L4_InOut_States : FB_PositionStateInOut;

    MR1L4_In : DUT_PositionState := (
        bUseRawCounts := TRUE,
        bMoveOk := TRUE,
        bValid := TRUE,
        sName := 'IN',
        nEncoderCount := 23615689,
        fDelta := 1000,
        fVelocity := 150);

    MR1L4_Out : DUT_PositionState := (
        bUseRawCounts := TRUE,
        bMoveOk := TRUE,
        bValid := TRUE,
        sName := 'OUT',
        nEncoderCount := 43989180,
        fDelta := 1000,
        fVelocity := 150);
END_VAR

//STATES
    MR1L3_SiC.stBeamParams.neVRange := F_eVExcludeRange(0, 1000) AND F_eVExcludeRange(13500, 90000);
    MR1L3_W.stBeamParams.neVRange := F_eVExcludeRange(0, 13000) AND F_eVExcludeRange(30000, 90000);

//M1L3 States with PMPS
    //Main.M1.bPowerSelf:=FALSE;
    fbMR1L3_Coating_States(
        bBPOkAutoReset := TRUE,
        bEnable := TRUE,
        stCoating1 := MR1L3_SiC,
        stCoating2 := MR1L3_W,
        fbArbiter:=GVL_PMPS.g_fbArbiter2,
        fbFFHWO:=GVL_PMPS.g_FastFaultOutput2 ,
        nTransitionAssertionID:= 16#FA71 ,
        nUnknownAssertionID:= 16#FA70 ,
        stMotionStage:=Main.M1);

//M1L3 States No State PMPS
    fbMR1L3_InOut_States(
        bEnable := TRUE,
        stIn := MR1L3_In,
        stOut := MR1L3_Out,
        stMotionStage := Main.M3);

//MR2L3 States No State PMPS
    fbMR2L3_Coating_States(
        bEnable := TRUE,
        stCoating1 := MR2L3_SiC,
        stCoating2 := MR2L3_W,
        stMotionStage:= Main.M13);

//MR1L4 States No State PMPS
    fbMR1L4_Coating_States(
        bEnable := TRUE,
        stCoating1 := MR1L4_SiC,
        stCoating2 := MR1L4_W,
        stMotionStage:= Main.M7);

    fbMR1L4_InOut_States(
        bEnable := TRUE,
        stIn := MR1L4_In,
        stOut := MR1L4_Out,
        stMotionStage := Main.M9);

END_PROGRAM

// ---- POUs/PRG_CoatingProtection.TcPOU
PROGRAM PRG_CoatingProtection
VAR
//M1
   fbM1 : FB_MirrorCoatingProtection := (
           sDevName:= 'XRT-M1',
        rFirstCoatingPosition:= 8611000,
        rFirstCoatingPositionTolerance:= 1000000,
        sFirstCoatingType:= 'SiC',
        rSecondCoatingPosition:= 18611000 ,
        rSecondCoatingPositionTolerance:= 1000000 ,
        sSecondCoatingType:= 'W',
        bAutoClear:= TRUE);

//M2
   fbM2 : FB_MirrorCoatingProtection := (
           sDevName:= 'XRT-M2',
        rFirstCoatingPosition:= 8496030,
        rFirstCoatingPositionTolerance:= 1000000,
        sFirstCoatingType:= 'SiC',
        rSecondCoatingPosition:= 18496030 ,
        rSecondCoatingPositionTolerance:= 1000000 ,
        sSecondCoatingType:= 'W',
        bAutoClear:= TRUE);

//M3
   fbM3 : FB_MirrorCoatingProtection := (
           sDevName:= 'XRT-M3',
        rFirstCoatingPosition:= 9279350,
        rFirstCoatingPositionTolerance:= 1000000,
        sFirstCoatingType:= 'SiC',
        rSecondCoatingPosition:= 19279350 ,
        rSecondCoatingPositionTolerance:= 1000000 ,
        sSecondCoatingType:= 'W',
        bAutoClear:= TRUE);



        // Fast Fault used when M1 and M2 are both in
         ffM1M2IN: FB_FastFault :=(
                    i_DevName := 'XRT-M1 and XRT-M2',
                    i_Desc := 'Fault occurs when both M1 and M2 are IN',
                    i_TypeCode := 16#602);
END_VAR

//M1
fbM1(
    bMirrorIn := (Main.nEncCntXupMR1L3 > 20210500) , // according to confluence -6 is nominal out position
    rCurrentEncoderPosition := Main.nEncCntYupMR1L3,
    neVRange := PMPS.PMPS_GVL.stCurrentBeamParameters.neVRange,
    nFirstCoatingBitmask:= F_eVExcludeRange(0, 1000) AND F_eVExcludeRange(13500, 90000),
    nSecondCoatingBitmask:= F_eVExcludeRange(0, 13000) AND F_eVExcludeRange(30000, 90000) ,
    FFO := GVL_PMPS.g_FastFaultOutput1);

//M2
//With M2 the same coating has different bit masks depending on the pitch
IF (Main.nEncCntPitchMR1L4 < 9616668 ) THEN//(HOMS2_Pitch.Stepper.stStatus.rActPosition < -400 ) THEN //MFX
    fbM2.nFirstCoatingBitmask:= F_eVExcludeRange(0, 1000) AND F_eVExcludeRange(13500, 90000);
    fbM2.nSecondCoatingBitmask:= F_eVExcludeRange(0, 13000) AND F_eVExcludeRange(30000, 90000);
ELSIF (Main.nEncCntPitchMR1L4 > 10129409 ) THEN// (HOMS2_Pitch.Stepper.stStatus.rActPosition > 600) THEN //MEC
    fbM2.nFirstCoatingBitmask:= F_eVExcludeRange(0, 1000) AND F_eVExcludeRange(25000, 90000);
    fbM2.nSecondCoatingBitmask:= F_eVExcludeRange(0, 13000) AND F_eVExcludeRange(30000, 90000);
ELSE // Anything else in the middle of the range
    fbM2.nFirstCoatingBitmask:= 0;
    fbM2.nSecondCoatingBitmask:= 0;
END_IF

fbM2(
    bMirrorIn := (Main.nEncCntXupMR1L4 < 25490840),
    rCurrentEncoderPosition := Main.nEncCntYupMR1L4,
    neVRange := PMPS.PMPS_GVL.stCurrentBeamParameters.neVRange,
    FFO := GVL_PMPS.g_FastFaultOutput1);

//M3
fbM3(
    bMirrorIn:=  fbM1.bMirrorIn, // When M1 is out, M3 is considered to be OUT
    rCurrentEncoderPosition := Main.nEncCntYupMR2L3,
    neVRange := PMPS.PMPS_GVL.stCurrentBeamParameters.neVRange,
    nFirstCoatingBitmask:= F_eVExcludeRange(0, 1000) AND F_eVExcludeRange(13500, 90000),
    nSecondCoatingBitmask:=  F_eVExcludeRange(0, 13000) AND F_eVExcludeRange(30000, 90000),
    FFO := GVL_PMPS.g_FastFaultOutput1);


// Evaluate M1 and M2 status
ffM1M2IN(
        i_xOK := NOT (fbM1.bMirrorIn AND fbM2.bMirrorIn),
        i_xAutoReset := TRUE,
        io_fbFFHWO:=GVL_PMPS.g_FastFaultOutput1);

END_PROGRAM

// ---- POUs/PRG_PMPS.TcPOU
PROGRAM PRG_PMPS
VAR
    bMR1L3_OUT_Veto: BOOL;
    fb_vetoArbiter: FB_VetoArbiter;
    ff2_ff1_link_vac: FB_FastFault := (i_xAutoReset := TRUE, i_DevName := 'FF2 to FF1 Link', i_Desc := 'This is virtual FF2 fault, Please check the faulting XRT Optics device', i_TypeCode := 16#9999);

    rtRemove: R_TRIG;
    bRemove :BOOL;
    bExist :BOOL;
    nReq : UDINT;
END_VAR


// PMPS Arbiter and FFO instantiation.
GVL_PMPS.g_fbArbiter1.AddRequest(16#5, PMPS_GVL.cstFullBeam, 'XRT HOMS');


GVL_PMPS.fbArbiterIO.i_bVeto := PMPS_GVL.stCurrentBeamParameters.aVetoDevices[PMPS.L_Stopper.ST1L0];
GVL_PMPS.fbArbiterIO(Arbiter := GVL_PMPS.g_fbArbiter1, fbFFHWO := GVL_PMPS.g_FastFaultOutput1);


bMR1L3_OUT_Veto := (( PRG_States.fbMR1L3_InOut_States.enumGet = ENUM_EpicsInOut.OUT) AND NOT ( PRG_States.fbMR1L3_InOut_States.enumGet = ENUM_EpicsInOut.IN));
fb_vetoArbiter(bVeto:=bMR1L3_OUT_Veto, // should Veto when MR1L3 is out of the beam
                HigherAuthority := GVL_PMPS.g_fbArbiter1,
                LowerAuthority := GVL_PMPS.g_fbArbiter2,
                FFO := GVL_PMPS.g_FastFaultOutput1);

GVL_PMPS.g_FastFaultOutput1.Execute(bAutoReset:=TRUE, i_xVeto:= PMPS_GVL.stCurrentBeamParameters.aVetoDevices[PMPS.L_Stopper.ST1L0]);
GVL_PMPS.g_FastFaultOutput2.Execute(bAutoReset:=TRUE, i_xVeto:= bMR1L3_OUT_Veto);


ff2_ff1_link_vac(
    io_fbFFHWO := GVL_PMPS.g_FastFaultOutput1,
    i_xOK := GVL_PMPS.g_FastFaultOutput2.q_xFastFaultOut);

// for testing and checking
bExist:= GVL_PMPS.g_fbArbiter1.CheckRequestInPool(nReq);
rtRemove(CLK:= bRemove);
if (rtRemove.Q) THEN
     GVL_PMPS.g_fbArbiter1.RemoveRequest(nReq);
END_IF

END_PROGRAM

// ---- GlobalTextList.TcGTLO
TEXTLIST GlobalTextList
  17 = '%.4f'
  18 = '%.4f V'
  22 = '%.6f um'
  51 = '%0.4f'
  52 = '%0.4f V'
  50 = '%0.6f um'
  7 = '%1.6f mm'
  10 = '%1.6f mm/s'
  44 = '%s'
  62 = '%t[ms]'
  9 = 'Absolute'
  8 = 'Absolute position'
  23 = 'Actual Position'
  21 = 'Actual Voltage'
  25 = 'Admin'
  12 = 'Axis Control'
  3 = 'Axis enabled'
  0 = 'Axis Status'
  35 = 'Closed Loop Control'
  54 = 'Couple'
  46 = 'Coupled'
  53 = 'Decouple'
  47 = 'Decoupled'
  16 = 'dX'
  1 = 'Enable Axis'
  34 = 'Enable Piezo'
  41 = 'Enable Primary Axis'
  5 = 'Error'
  40 = 'Expert Mode'
  49 = 'For controlling coupled movement'
  57 = 'Gantry Controls'
  45 = 'Gantry Mode'
  33 = 'Ki'
  32 = 'Kp'
  55 = 'Label'
  2 = 'Minus limit switch is hit'
  28 = 'None'
  27 = 'Operator'
  56 = 'Overall System Controls'
  38 = 'Pitch Manual Mode'
  4 = 'Plus limit switch is hit'
  42 = 'Primary Axis'
  39 = 'Puts the pitch control function block into manual mode. In manual mode the piezo and stepper movements are completely independent of one another and no coordinated actions take place. Limit switches are still respected.'
  11 = 'Relative'
  24 = 'Requested Position'
  19 = 'Requested Voltage'
  6 = 'Reset error.'
  43 = 'Secondary Axis'
  26 = 'Service'
  20 = 'Set Voltage'
  61 = 'Setpoint Voltage'
  13 = 'Simulation Axis 1'
  60 = 'Simulator Gantry Controls'
  37 = 'Start'
  31 = 'Start absolute move'
  48 = 'Virtual Axis'
  36 = 'Voltage Control'
  29 = 'Voltage mode'
  30 = 'Voltage Mode'
  15 = 'X'
  58 = 'X Gantry Controls'
  14 = 'Y'
  59 = 'Y Gantry Controls'
END_TEXTLIST

// ---- VISUs/GantryControls.TcVIS
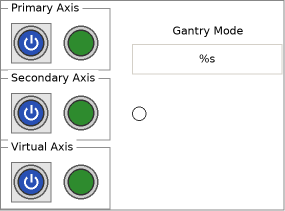
VISUALIZATION GantryControls  // 285x211
VAR_IN_OUT
	Gantry	:	HOMS_Gantry;
END_VAR
    GroupBox (0,0 110x70), "Primary Axis"
        PowerSwitch (11,23 40x40), variable: Gantry.PAxis.xEnable, behaviour: TOGGLE, style: Switch-PowerSwitch-Blue
        Lamp1 (61,23 40x40), variable: NOT Gantry.PAxis.stAxis.Status.Disabled, style: Lamp-Lamp1-Green
    GroupBox (0,70 110x70), "Secondary Axis"
        PowerSwitch (11,23 40x40), variable: Gantry.SAxis.xEnable, behaviour: TOGGLE, style: Switch-PowerSwitch-Blue
        Lamp1 (61,23 40x40), variable: NOT Gantry.SAxis.stAxis.Status.Disabled, style: Lamp-Lamp1-Green
    Textfield (132,44 150x30), "%s", text variable: Gantry.Mode
    Label (133,16 150x30), "Gantry Mode"
    RadioButton (130,82 150x63), variable: Gantry.ModeReq, input disabled if: Gantry.PAxis.stAxis.Status.Moving
        Areas[0]: Text=Coupled
        Areas[1]: Text=Decoupled
    GroupBox (0,139 110x70), "Virtual Axis", tooltip "For controlling coupled movement"
        PowerSwitch (11,23 40x40), variable: Gantry.VAxis.xEnable, behaviour: TOGGLE, style: Switch-PowerSwitch-Blue
        Lamp1 (61,23 40x40), variable: Gantry.SAxis.stAxis.Status.Coupled AND NOT Gantry.PAxis.stAxis.Status.Disabled AND NOT Gantry.SAxis.stAxis.Status.Disabled, style: Lamp-Lamp1-Green
END_VISUALIZATION

// ---- VISUs/Visualization.TcVIS
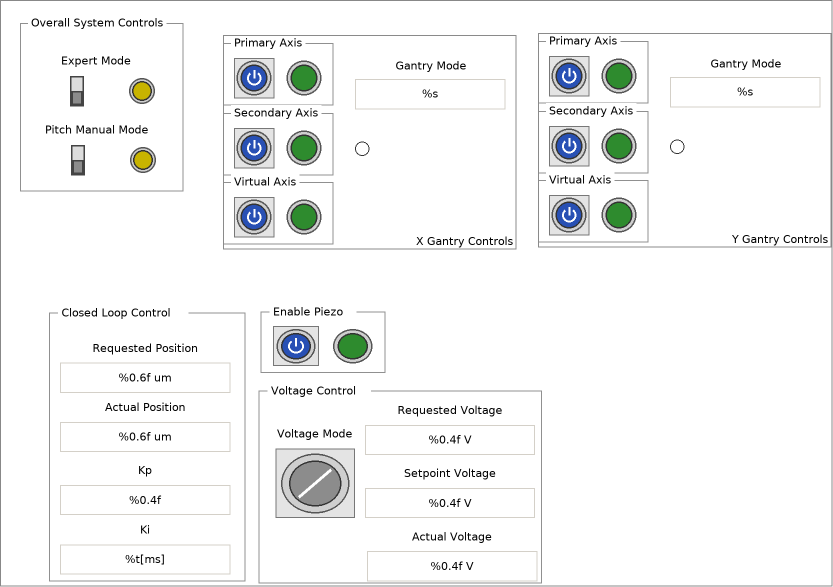
VISUALIZATION Visualization  // 833x587
    Frame (223,35 293x214), "X Gantry Controls"
        shows GantryControls(Gantry := XGantry)
    GroupBox (20,15 163x176), "Overall System Controls"
        Group (17,31 120x60)
            DipSwitch (0,30 80x30), tooltip "Puts the pitch control function block into manual mode. In manual mode the piezo and stepper movements are completely independent of one another and no coordinated actions take place. Limit switches are still respected.", variable: MAIN.ExpertMode, behaviour: TOGGLE, style: Switch-DipSwitch-Gray
            Label (3,0 112x30), "Expert Mode"
            Lamp1 (90,30 30x30), variable: MAIN.ExpertMode, style: Lamp-Lamp1-Yellow
        Group (18,100 120x60)
            DipSwitch (0,30 80x30), tooltip "Puts the pitch control function block into manual mode. In manual mode the piezo and stepper movements are completely independent of one another and no coordinated actions take place. Limit switches are still respected.", variable: MAIN.PitchManualMode, behaviour: TOGGLE, style: Switch-DipSwitch-Gray
            Label (3,0 112x30), "Pitch Manual Mode"
            Lamp1 (90,30 30x30), variable: MAIN.PitchControl.ManualMode, style: Lamp-Lamp1-Yellow
    Frame (31,284 513x301)
        shows PiezoControls(Piezo := gPitch.Piezo, ActPos := gPitch.Stepper)
    Frame (538,33 293x214), "Y Gantry Controls"
        shows GantryControls(Gantry := YGantry)
END_VISUALIZATION

// ---- VISUs/PiezoControls.TcVIS
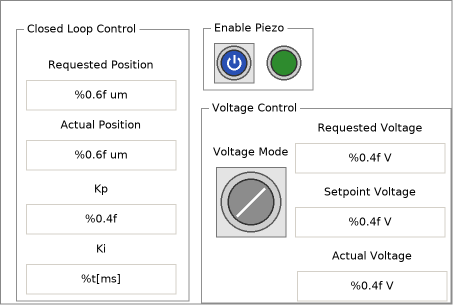
VISUALIZATION PiezoControls  // 453x305
VAR_IN_OUT
	Piezo	:	ST_PiezoAxis;
	ActPos	:	ST_HOMSStepper;
END_VAR
    GroupBox (203,20 110x70), "Enable Piezo"
        PowerSwitch (11,23 40x40), variable: Piezo.xEnable, behaviour: TOGGLE, style: Switch-PowerSwitch-Blue
        Lamp1 (61,23 40x40), variable: Piezo.xEnable and NOT Piezo.xError, style: Lamp-Lamp1-Green
    GroupBox (16,21 173x280), "Closed Loop Control"
        Textfield (10,59 150x30), "%0.6f um", text variable: Piezo.rReqAbsPos
            OnMouseClick: write the text variable via Default
        Textfield (10,119 150x30), "%0.6f um", text variable: ActPos.stAxis.NcToPlc.ActPos
        Label (10,89 150x30), "Actual Position"
        Label (10,29 150x30), "Requested Position"
        Textfield (10,183 150x30), "%0.4f", text variable: Piezo.stPIParams.fKp
            OnMouseClick: write the text variable via Default
        Textfield (10,243 150x30), "%t[ms]", text variable: Piezo.stPIParams.tTn
            OnMouseClick: write the text variable via Edit
        Label (10,153 150x30), "Kp"
        Label (10,213 150x30), "Ki"
    GroupBox (201,100 250x203), "Voltage Control"
        Textfield (94,43 150x30), "%0.4f V", text variable: Piezo.rReqVoltage
            OnMouseClick: write the text variable via Default
        Label (94,13 150x30), "Requested Voltage"
        Textfield (94,107 150x30), "%0.4f V", text variable: Piezo.rSetVoltage
        Label (94,77 150x30), "Setpoint Voltage"
        RotarySwitch (15,67 70x70), tooltip "Voltage mode", variable: Piezo.xVoltageMode, behaviour: TOGGLE, style: Switch-RotarySwitch-Gray
        Label (5,37 90x30), "Voltage Mode"
        Label (96,141 150x30), "Actual Voltage"
        Textfield (96,171 150x30), "%0.4f V", text variable: Piezo.rActVoltage
END_VISUALIZATION
